TYPE ST_CanHeader :
STRUCT
	nCobid: DWORD; // User level Cobid, use functions to handle bit mapping to CAN interface process data.
	bExtendedAddress: BOOL;// does nothing with 11bit version. Incorrectly 'cleared' does not cause errors and is automatically fixed.
	bRTR: BOOL; // Remote transmission request
	nMsgLength: UINT; // number of bytes in CAN message, values 0-8
END_STRUCT
END_TYPE

(* stored: Version 1.1.0.1, ProductVersion 3.1.4024.12
   DUT ST_CanHeader: Id {cb3812b6-57a6-05a5-032e-846a90d5b8f0} *)
